{attribute 'linkalways'} 
{attribute 'no_explicit_call' := 'This FB is a CLASS and must be accessed using methods or properties'}
{attribute 'enable_dynamic_creation'}
FUNCTION_BLOCK _ETcVnContainerExportFormat EXTENDS EnumDatatypeBase
VAR
	localData : ETcVnContainerExportFormat;
	activeData : REFERENCE TO ETcVnContainerExportFormat;
	enumBaseDatatype : _UINT(localData);
END_VAR

METHOD PRIVATE AddLocalEnumeration
VAR_INPUT
	Enumeration : T_MAXSTRING;
	Value : ETcVnContainerExportFormat;
END_VAR
AddEnumeration(Enumeration, Value);
END_METHOD

PROPERTY PUBLIC Address : PVOID
GET
Address := ADR(activeData);
END_GET
END_PROPERTY

METHOD PUBLIC ClearReference
VAR_INPUT
END_VAR
activeData REF= localData;
SetBaseDatatypeReference();
END_METHOD

METHOD PUBLIC Clone : I_Datatype
VAR
    pClone : POINTER TO _ETcVnContainerExportFormat;
END_VAR
pClone := __NEW(_ETcVnContainerExportFormat(InitialValue := Value));
Clone := pClone^;
END_METHOD

METHOD FB_init : BOOL
VAR_INPUT
	bInitRetains : BOOL; // if TRUE, the retain variables are initialized (warm start / cold start)
	bInCopyCode : BOOL;  // if TRUE, the instance afterwards gets moved into the copy code (online change)
	InitialValue : ETcVnContainerExportFormat;
END_VAR
localData := InitialValue;
AddBaseDatatype(enumBaseDatatype);
ClearReference();

AddLocalEnumeration('TCVN_CEF_XML', ETcVnContainerExportFormat.TCVN_CEF_XML);
AddLocalEnumeration('TCVN_CEF_XML_SERIALIZED', ETcVnContainerExportFormat.TCVN_CEF_XML_SERIALIZED);
AddLocalEnumeration('TCVN_CEF_CSV', ETcVnContainerExportFormat.TCVN_CEF_CSV);
AddLocalEnumeration('TCVN_CEF_BINARY', ETcVnContainerExportFormat.TCVN_CEF_BINARY);
END_METHOD

PROPERTY PUBLIC Identifier : T_MAXSTRING
GET
Identifier := 'ETcVnContainerExportFormat';
END_GET
END_PROPERTY

METHOD IsEnumeratorValueEqual : BOOL
VAR_INPUT
	Enumerator : I_KeyValueForwardEnumerator;
END_VAR
VAR
	storedValue : ETcVnContainerExportFormat;
END_VAR
IF NOT Enumerator.TryGet(storedValue) THEN
	RETURN;
END_IF

IsEnumeratorValueEqual := storedValue = activeData;
END_METHOD

METHOD PUBLIC MakeReferenceTo
VAR_INPUT
	ReferenceTarget : REFERENCE TO ETcVnContainerExportFormat;
END_VAR
activeData REF= ReferenceTarget;
SetBaseDatatypeReference();
END_METHOD

METHOD PROTECTED SetBaseDatatypeReference
VAR_INPUT
END_VAR
enumBaseDatatype.MakeReferenceTo(activeData);
END_METHOD

PROPERTY PUBLIC Size : UDINT
GET
Size := SIZEOF(activeData);
END_GET
END_PROPERTY

METHOD TryMakeReferenceTo : BOOL
VAR_INPUT
	Target : I_Datatype;
END_VAR
VAR
	targetAsEnum : I_EnumDatatype;
	pTargetData : POINTER TO ETcVnContainerExportFormat;
END_VAR
IF NOT Target.TryResolveAsEnumDatatype(targetAsEnum) THEN
	RETURN;
END_IF

IF targetAsEnum.Identifier <> Identifier THEN
	RETURN;
END_IF

pTargetData := Target.Address;
activeData REF= pTargetData^;
SetBaseDatatypeReference();
TryMakeReferenceTo := TRUE;
END_METHOD

PROPERTY PUBLIC Value : ETcVnContainerExportFormat
GET
Value := activeData;
END_GET
SET
activeData := Value;
END_SET
END_PROPERTY

END_FUNCTION_BLOCK

(* stored: Version 1.1.0.1
   POU _ETcVnContainerExportFormat: Id {ad122f32-6f04-4c22-ac1a-7f7d25abda77}, SpecialFunc None
   Folder Constructor: Id {eb2149f3-0ec7-4efd-a2f0-4b7543b8f21b}
   Folder Private: Id {1caa6af0-4d01-4037-98a4-900fca5ab527}
   Folder Protected: Id {d6be9eee-edc9-40be-aa22-b48bcfa011eb}
   Method AddLocalEnumeration: Id {f2d4f5e0-5798-42f0-b25a-4f1ded853c47}
   Property Address: Id {dcb4c5a8-6d48-4239-b6e3-3c4925cb2a0e}
   Get Get: Id {5b563842-a4e4-4163-9a3f-d157cd2b150d}
   Method ClearReference: Id {2b6f5ad0-f7d7-4c80-b02e-9cc3279b0694}
   Method Clone: Id {5a666300-030d-4f82-a3dc-a8c607ff0e6f}
   Method FB_init: Id {084bc5f4-37d6-493b-9d69-d7732b2c5985}
   Property Identifier: Id {6476a521-3782-4236-b2f2-8c2841baef97}
   Get Get: Id {fd0c988b-ea12-4461-9c5e-7e1f2c5bd506}
   Method IsEnumeratorValueEqual: Id {f402fc5d-c367-4e20-9a58-ee1bc6b852b8}
   Method MakeReferenceTo: Id {8691a0ef-be60-430f-8c50-002d97a9553a}
   Method SetBaseDatatypeReference: Id {c85d9477-ee46-4e77-8b2b-51519568ab9f}
   Property Size: Id {cc383bec-c0cf-4552-8d82-44edb679bf4c}
   Get Get: Id {22e84e3b-a746-43cf-8b3b-ab29c293de65}
   Method TryMakeReferenceTo: Id {2652f858-98ce-4d5f-bf53-ca01e917915f}
   Property Value: Id {19c2792e-eaa7-44d8-8788-99ff1d7e6240}
   Get Get: Id {84d0ef08-fd18-451d-bbee-e470a5504347}
   Set Set: Id {43d16fa5-d853-4bae-8ba4-e955f309e825} *)
